FUNCTION_BLOCK AXE_plant_FV
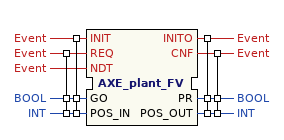
  EVENT_INPUT
    INIT WITH GO, POS_IN;
    REQ WITH GO, POS_IN;
    NDT;
  END_EVENT
  EVENT_OUTPUT
    INITO WITH PR, POS_OUT;
    CNF WITH PR, POS_OUT;
  END_EVENT
  VAR_INPUT
    GO : BOOL;
    POS_IN : INT;
  END_VAR
  VAR_OUTPUT
    PR : BOOL;
    POS_OUT : INT;
  END_VAR
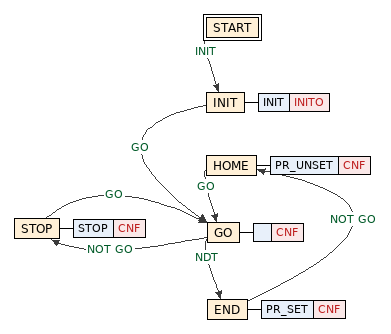
  EC_STATES
    START;
    HOME : PR_UNSET -> CNF;
    GO : -> CNF;
    END : PR_SET -> CNF;
    STOP : STOP -> CNF;
    INIT : INIT -> INITO;
  END_STATES
  EC_TRANSITIONS
    HOME TO GO := GO;
    STOP TO GO := GO;
    GO TO STOP := NOT GO;
    GO TO END := NDT;
    END TO HOME := NOT GO;
    START TO INIT := INIT;
    INIT TO GO := GO;
  END_TRANSITIONS
  ALGORITHM INIT IN ST:
PR := FALSE;
  END_ALGORITHM
  ALGORITHM PR_SET IN ST:
PR := TRUE;
POS_OUT := POS_IN;
  END_ALGORITHM
  ALGORITHM STOP IN ST:
PR := FALSE;
POS_OUT := 5;
  END_ALGORITHM
  ALGORITHM PR_UNSET IN ST:
PR := FALSE;
  END_ALGORITHM
END_FUNCTION_BLOCK
